{attribute 'qualified_only'}
{attribute 'strict'}
{attribute 'to_string'}
TYPE E_INSTANCE_STATE :
(
	INVALID,
  INIT,
  DISABLED,
  DETECT_IN_LIST,
  ENABLED,
  WORKING,
  FINISH
);
END_TYPE

(* stored: Version 1.1.0.1
   DUT E_INSTANCE_STATE: Id {835bcac6-d9c6-4e45-b545-3a98d3dea6a0} *)
